{attribute 'qualified_only'}
VAR_GLOBAL
	test: BOOL;
END_VAR

(* stored: Version 1.1.0.1, ProductVersion 3.1.4024.11
   GVL DataConfig: Id {c5482dc7-5fc1-41fb-bde1-3036a029dc4e} *)
